PROGRAM P_Dimmers_Broadcast
VAR
	fbDALIV2Dimmer2Switch_RB1		: FB_DALIV2Dimmer2Switch;
	nActualLEvelMasterDev_1			: BYTE;
	bBusy_1							: BOOL;
	bError_1						: BOOL;
	nErrorId_1						: UDINT;
	
	
	fbDALIV2Dimmer2Switch_RB2		: FB_DALIV2Dimmer2Switch;
	nActualLEvelMasterDev_2			: BYTE;
	bBusy_2							: BOOL;
	bError_2						: BOOL;
	nErrorId_2						: UDINT;
	
	
	fbDALIV2Dimmer2Switch_RB3		: FB_DALIV2Dimmer2Switch;
	nActualLEvelMasterDev_3			: BYTE;
	bBusy_3							: BOOL;
	bError_3						: BOOL;
	nErrorId_3						: UDINT;
END_VAR

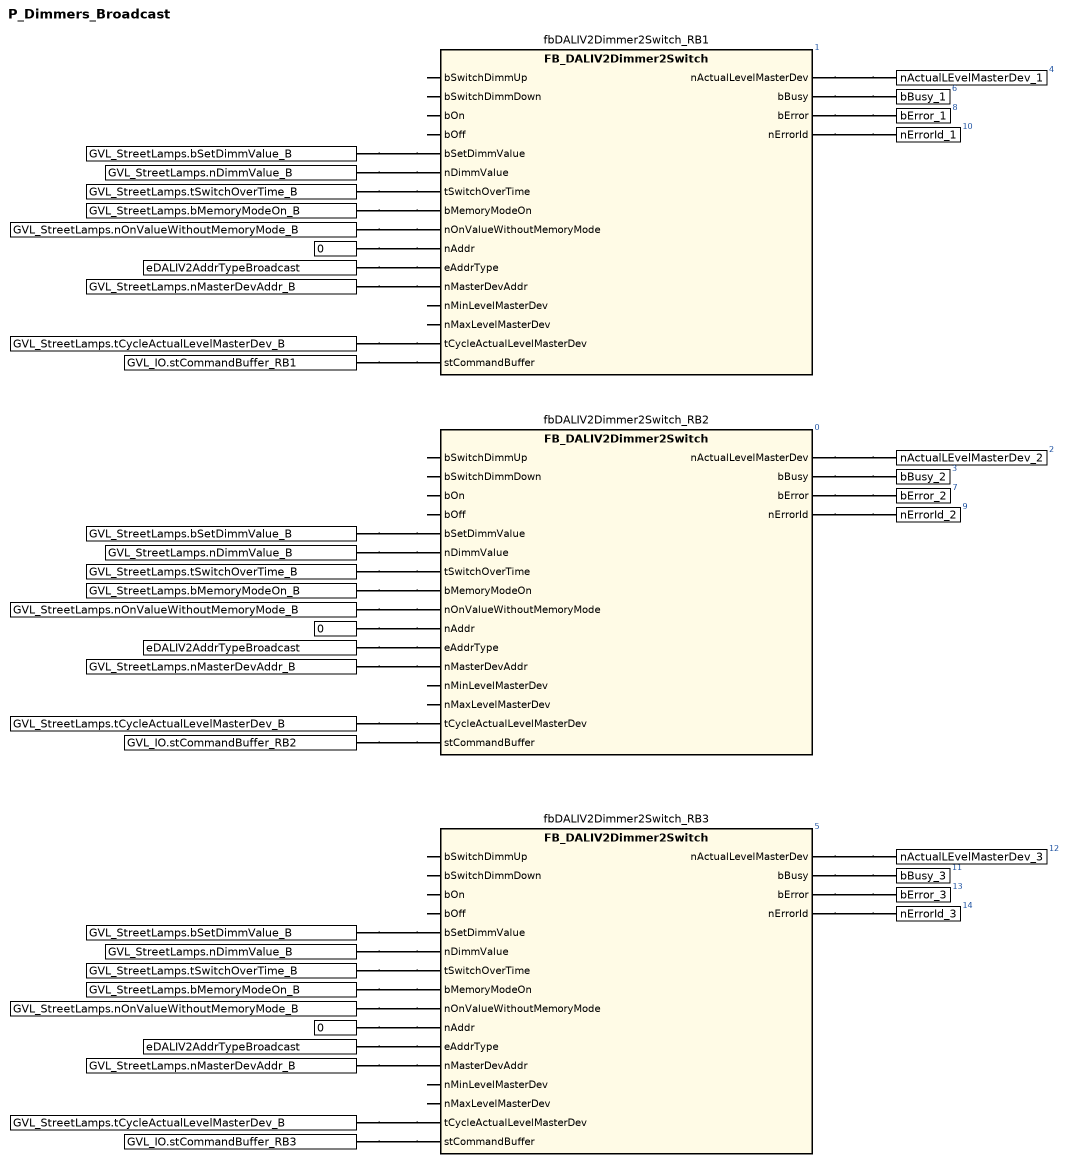
fbDALIV2Dimmer2Switch_RB2(
    bSetDimmValue := GVL_StreetLamps.bSetDimmValue_B,
    nDimmValue := GVL_StreetLamps.nDimmValue_B,
    tSwitchOverTime := GVL_StreetLamps.tSwitchOverTime_B,
    bMemoryModeOn := GVL_StreetLamps.bMemoryModeOn_B,
    nOnValueWithoutMemoryMode := GVL_StreetLamps.nOnValueWithoutMemoryMode_B,
    nAddr := 0,
    eAddrType := eDALIV2AddrTypeBroadcast,
    nMasterDevAddr := GVL_StreetLamps.nMasterDevAddr_B,
    tCycleActualLevelMasterDev := GVL_StreetLamps.tCycleActualLevelMasterDev_B,
    stCommandBuffer := GVL_IO.stCommandBuffer_RB2); // FB_DALIV2Dimmer2Switch
fbDALIV2Dimmer2Switch_RB1(
    bSetDimmValue := GVL_StreetLamps.bSetDimmValue_B,
    nDimmValue := GVL_StreetLamps.nDimmValue_B,
    tSwitchOverTime := GVL_StreetLamps.tSwitchOverTime_B,
    bMemoryModeOn := GVL_StreetLamps.bMemoryModeOn_B,
    nOnValueWithoutMemoryMode := GVL_StreetLamps.nOnValueWithoutMemoryMode_B,
    nAddr := 0,
    eAddrType := eDALIV2AddrTypeBroadcast,
    nMasterDevAddr := GVL_StreetLamps.nMasterDevAddr_B,
    tCycleActualLevelMasterDev := GVL_StreetLamps.tCycleActualLevelMasterDev_B,
    stCommandBuffer := GVL_IO.stCommandBuffer_RB1); // FB_DALIV2Dimmer2Switch
nActualLEvelMasterDev_2 := fbDALIV2Dimmer2Switch_RB2.nActualLevelMasterDev;
bBusy_2 := fbDALIV2Dimmer2Switch_RB2.bBusy;
nActualLEvelMasterDev_1 := fbDALIV2Dimmer2Switch_RB1.nActualLevelMasterDev;
fbDALIV2Dimmer2Switch_RB3(
    bSetDimmValue := GVL_StreetLamps.bSetDimmValue_B,
    nDimmValue := GVL_StreetLamps.nDimmValue_B,
    tSwitchOverTime := GVL_StreetLamps.tSwitchOverTime_B,
    bMemoryModeOn := GVL_StreetLamps.bMemoryModeOn_B,
    nOnValueWithoutMemoryMode := GVL_StreetLamps.nOnValueWithoutMemoryMode_B,
    nAddr := 0,
    eAddrType := eDALIV2AddrTypeBroadcast,
    nMasterDevAddr := GVL_StreetLamps.nMasterDevAddr_B,
    tCycleActualLevelMasterDev := GVL_StreetLamps.tCycleActualLevelMasterDev_B,
    stCommandBuffer := GVL_IO.stCommandBuffer_RB3); // FB_DALIV2Dimmer2Switch
bBusy_1 := fbDALIV2Dimmer2Switch_RB1.bBusy;
bError_2 := fbDALIV2Dimmer2Switch_RB2.bError;
bError_1 := fbDALIV2Dimmer2Switch_RB1.bError;
nErrorId_2 := fbDALIV2Dimmer2Switch_RB2.nErrorId;
nErrorId_1 := fbDALIV2Dimmer2Switch_RB1.nErrorId;
bBusy_3 := fbDALIV2Dimmer2Switch_RB3.bBusy;
nActualLEvelMasterDev_3 := fbDALIV2Dimmer2Switch_RB3.nActualLevelMasterDev;
bError_3 := fbDALIV2Dimmer2Switch_RB3.bError;
nErrorId_3 := fbDALIV2Dimmer2Switch_RB3.nErrorId;

END_PROGRAM

(* stored: Version 1.1.0.1, ProductVersion 3.1.4024.5
   POU P_Dimmers_Broadcast: Id {b525ded5-5d3f-48ca-a33a-633e19d8cc5f}, SpecialFunc None *)
